KUKA KRL data list: mcv_main.dat

&ACCESS RVP
&REL 3
&PARAM DISKPATH = KRC:\R1\Program\MCV
DEFDAT mcv_main PUBLIC

  ; Home position
  DECL E6AXIS XHOME = {A1 0.0, A2 -90.0, A3 90.0, A4 0.0, A5 0.0, A6 0.0, E1 0.0, E2 0.0, E3 0.0, E4 0.0, E5 0.0, E6 0.0}

  ; External declarations
  EXTERNAL mcv_milling()

ENDDAT
